SREFP 2 C00641 BC00641  +REFP EC00641
MACRO1 MJ#(0) ARGF0
ARCON
SMOVL C00642 BC00642 V=10.0  +MOVJ EC00642
SMOVL C00643 BC00643 V=10.0  +MOVJ EC00643
SMOVL C00644 BC00644 V=10.0  +MOVJ EC00644
ARCOF
MOVL C00645 BC00645 V=400.0  +MOVJ EC00645 VJ=100.00
MOVL C00646 BC00646 V=1000.0  +MOVJ EC00646 VJ=100.00
MOVL C00647 BC00647 V=1000.0  +MOVJ EC00647 VJ=100.00
MOVJ C00648 BC00648 VJ=100.00  +MOVJ EC00648 VJ=100.00
MOVJ C00649 BC00649 VJ=100.00  +MOVJ EC00649 VJ=100.00
MOVJ C00650 BC00650 VJ=100.00  +MOVJ EC00650 VJ=100.00
MOVJ C00651 BC00651 VJ=100.00  +MOVJ EC00651 VJ=100.00
'68,69
MOVJ C00652 BC00652 VJ=100.00  +MOVJ EC00652 VJ=100.00
'Path W1655
SFTOF3D
SFTON3D P030
MOVJ C00653 BC00653 VJ=100.00  +MOVJ EC00653 VJ=100.00
SMOVL C00654 BC00654 V=100.0  +MOVJ EC00654
SMOVL C00655 BC00655 V=100.0 PL=0  +MOVJ EC00655
SREFP 1 C00656 BC00656  +REFP EC00656
SREFP 2 C00657 BC00657  +REFP EC00657
MACRO1 MJ#(0) ARGF0
ARCON
SFTON3D P029
SMOVL C00658 BC00658 V=10.0  +MOVJ EC00658
SFTON3D P028
SMOVL C00659 BC00659 V=10.0  +MOVJ EC00659
ARCOF
SMOVL C00660 BC00660 V=400.0  +MOVJ EC00660
SMOVL C00661 BC00661 V=1000.0  +MOVJ EC00661
SFTOF3D
MOVJ C00662 BC00662 VJ=100.00  +MOVJ EC00662 VJ=100.00
MOVJ C00663 BC00663 VJ=100.00  +MOVJ EC00663 VJ=100.00
COMM 'Path W1656
COMM SFTOF3D
COMM SFTON3D P031
COMM MOVJ C00664 BC00664 VJ=100.00  +MOVJ EC00664 VJ=100.00
COMM SMOVL C00665 BC00665 V=100.0  +MOVJ EC00665
COMM SMOVL C00666 BC00666 V=100.0 PL=0  +MOVJ EC00666
COMM SREFP 1 C00667 BC00667  +REFP EC00667
COMM SREFP 2 C00668 BC00668  +REFP EC00668
COMM MACRO1 MJ#(0) ARGF0
COMM ARCON
COMM SMOVL C00669 BC00669 V=10.0  +MOVJ EC00669
COMM SMOVL C00670 BC00670 V=10.0  +MOVJ EC00670
COMM SMOVL C00671 BC00671 V=10.0  +MOVJ EC00671
COMM ARCOF
COMM SMOVL C00672 BC00672 V=400.0  +MOVJ EC00672
COMM SMOVL C00673 BC00673 V=1000.0  +MOVJ EC00673
SFTOF3D
MOVJ C00674 BC00674 VJ=100.00  +MOVJ EC00674 VJ=100.00
MOVJ C00675 BC00675 VJ=100.00  +MOVJ EC00675 VJ=100.00
MOVJ C00676 BC00676 VJ=0.78  +MOVJ EC00676 VJ=0.78
'Down
END
